(* Logix 5000 project; controller TBEN_Lx_8IOL_AOI_V0_2 vendor 1 type 14 code 176 rev 32.11; software revision 32.00; part 8 of 11 *)
(* tags used below, declared in another part *)
   Process_Input_Data : Generic_173_Words;
   Process_Output_Data : Generic_131_Words;
(* IOLService_ISDU, continued *)

ROUTINE Prescan   (* ladder *)
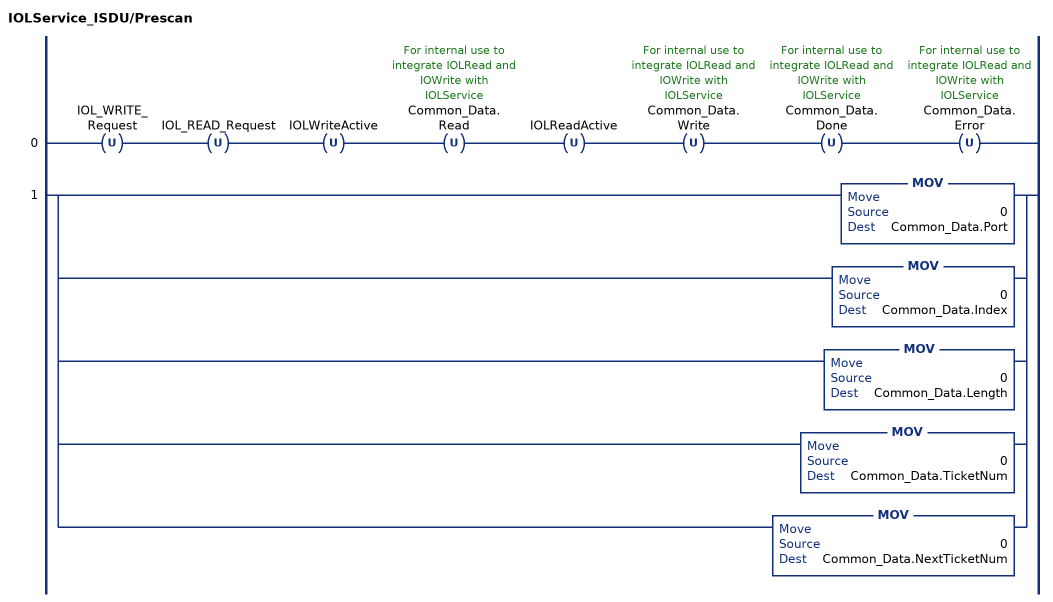
   0: OTU(IOL_WRITE_Request)OTU(IOL_READ_Request)OTU(IOLWriteActive)OTU(Common_Data.Read)OTU(IOLReadActive)OTU(Common_Data.Write)OTU(Common_Data.Done)OTU(Common_Data.Error);
   1: [MOV(0,Common_Data.Port) ,MOV(0,Common_Data.Index) ,MOV(0,Common_Data.Length) ,MOV(0,Common_Data.TicketNum) ,MOV(0,Common_Data.NextTicketNum) ];
END_ROUTINE
END_ADD_ON_INSTRUCTION

ADD_ON_INSTRUCTION TBEN_Lx_8IOL_AOI   (* revision 0.3 Unreleased, vendor Turck, ExecutePrescan *)
// AOI specific to TBEN-Lx-8IOL devices. It requires the  Input, Output, Config tags from the catalog file.
// Revision note:
// V0_1 Initial Approach
// V0_2 Cleaning Up
// V0_3 Changes to process Data
// Help:
// IOL_Service - used with Turck BL20, BL67, BLC and TBEN IOLink masters to process requests from IOL_ReadString, IOL_WriteString, IOL_ReadData and IOL_WriteData AOI's.
// Status	Description
// 0	Operation completed successfully
// 	Status = 100 - 102, Ethernet IP MSG instruction errors - check communication parameters
// 100	IOL_SendMSG completed with error, check communication parameters
// 101	IOL_RecevieMSG completed with error, check communication parameters
// 110	IOL_Service Retry Limit exceeded
// 111	Slot specified not an IOLink master
// 	Status = 1000 to 1255, no response from device, connection error
// 1016	Device not connected or Port not configured as IOLink port
// 	Status = 2000 to 2255,  device response indicates error
// 2000	Device error, no details
// 2017	Device error, Index not available
// 2018	Device error, Subindex not available
// 2032	Device error, Service temporarily not available
// 2033	Device error, Service temporarily not available - local control
// 2034	Device error, Service temporarily not available - device control
// 2035	Device error, Index not writeable
// 2048	Device error, Parameter value out of range
// 2049	Device error, Parameter value above limit
// 2050	Device error, Parameter value below limit
// 2051	Device error, Parameter value length overrun (check IOLWrite precision/string length)
// 2052	Device error, Parameter value length underrun (check IOLWrite precision/string length)
// 2053	Device error, Function not available
// 2054	Device error, Function temporarily not available
// 2064	Device error, Parameter set invalid
// 2065	Device error, Inconsistent parameter set
// 2130	Device error, Application not ready
// 	Status = 3000 to 3255,   device response indicates vendor specific error
// 3000	Vendor specific error, no details
// 3001	Vendor specific error, vendor specific error number
// 3255	Vendor specific error, vendor specific error number
// 	Status = 7000 to 7255,  IOL-M Error Codes
// 7000	Unexpected write request instead of read request
// 7001	Decode error
// 7002	Port occupied by another task
// 	Status = 8000 to 8255,  IOL-M Error Codes
// 8000	Timeout when IOL-Ds or IOL-M ports are busy
// 8001	IOL Index out of range
// 8002	Port address greater than maximum
// 8003	Port function not supported
VAR_IN_OUT
   Common_Data : Turck_IOLink_Common_Data; {required}
        .SendData[1]   // For internal use to integrate IOLRead and IOLWrite with IOLService
   IOL_Read_MSG : MESSAGE; {required}
   IOL_Write_MSG : MESSAGE; {required}
   TBEN_I_DATA : INT[173]; {required}   // Input Data from IO Block
   TBEN_O_DATA : INT[131]; {required}   // Output Data to IO Block
   TBEN_C_DATA : SINT[160]; {required}
END_VAR
VAR_OUTPUT
   DXP1_OUT : BOOL; {visible}
   DXP3_OUT : BOOL; {visible}
   DXP5_OUT : BOOL; {visible}
   DXP7_OUT : BOOL; {visible}
   IOLDevice_PORT1 : BOOL; {visible}
   IOLDevice_PORT2 : BOOL; {visible}
   IOLDevice_PORT3 : BOOL; {visible}
   IOLDevice_PORT4 : BOOL; {visible}
   IOLDevice_PORT5 : BOOL; {visible}
   IOLDevice_PORT6 : BOOL; {visible}
   IOLDevice_PORT7 : BOOL; {visible}
   IOLDevice_PORT8 : BOOL; {visible}
END_VAR
VAR_INPUT
   IOL0_DI : BOOL; {visible}
   DXP1_IN : BOOL; {visible}
   IOL2_DI : BOOL; {visible}
   DXP3_IN : BOOL; {visible}
   IOL4_DI : BOOL; {visible}
   DXP5_IN : BOOL; {visible}
   IOL6_DI : BOOL; {visible}
   DXP7_IN : BOOL; {visible}
   IOL8_DI : BOOL; {visible}
   IOL10_DI : BOOL; {visible}
   IOL12_DI : BOOL; {visible}
   IOL14_DI : BOOL; {visible}
   PORT1_Mode_IOL_or_DI : BOOL;   // 0: IO-LINK without validation 1: Port is set to DI (Power Cycle or Module Inhibit cycle require)
   PORT2_Mode_IOL_or_DI : BOOL;   // 0: IO-LINK without validation 1: Port is set to DI (Power Cycle or Module Inhibit cycle require)
   PORT3_Mode_IOL_or_DI : BOOL;   // 0: IO-LINK without validation 1: Port is set to DI (Power Cycle or Module Inhibit cycle require)
   PORT4_Mode_IOL_or_DI : BOOL;   // 0: IO-LINK without validation 1: Port is set to DI (Power Cycle or Module Inhibit cycle require)
   PORT5_Mode_IOL_or_DI : BOOL;   // 0: IO-LINK without validation 1: Port is set to DI (Power Cycle or Module Inhibit cycle require)
   PORT6_Mode_IOL_or_DI : BOOL;   // 0: IO-LINK without validation 1: Port is set to DI (Power Cycle or Module Inhibit cycle require)
   PORT7_Mode_IOL_or_DI : BOOL;   // 0: IO-LINK without validation 1: Port is set to DI (Power Cycle or Module Inhibit cycle require)
   PORT8_Mode_IOL_or_DI : BOOL;   // 0: IO-LINK without validation 1: Port is set to DI (Power Cycle or Module Inhibit cycle require)
   DisableOutput_DXP1 : BOOL;
   DisableOutput_DXP3 : BOOL;
   DisableOutput_DXP5 : BOOL;
   DisableOutput_DXP7 : BOOL;
END_VAR
VAR_OUTPUT
   Device_Restart_Required : BOOL; {visible}
END_VAR
VAR
   IOLReadActive : BOOL;
   IOLWriteActive : BOOL;
   RetryCount : DINT;
   IOL_Error_Count : DINT; {access None}
   IOLReset_ONS : BOOL; {access None}
   ER1 : BOOL; {access None}
   ER2 : BOOL; {access None}
   tempReceiveData : SINT[255]; {access None}
   Generate_Status : BOOL; {access None}
   ABS_RD_0 : INT; {access None}
   ABS_RD_1 : INT; {access None}
   ABS_RD_2 : INT; {access None}
   ABS_RD_3 : INT; {access None}
   tempSendData : SINT[145]; {access None}
   IOL_READ_Request : BOOL; {access None}
   IOL_WRITE_Request : BOOL; {access None}
   StartupDone : BOOL; {access None}
   Done : BOOL; {access None}
   Error : BOOL; {access None}
   Active : BOOL; {access None}
   Pending : BOOL; {access None}
   Pending_or_Active : BOOL; {access None}
   StartupCount : SINT; {access None}
   DoneCount : SINT; {access None}
   MyTicketNum : INT; {access None}
   Update_Data : BOOL; {access None}
   Read_ONS : BOOL; {access None}
   ReadRequest : BOOL; {access None}
   Prev_Input_Data_Valids : INT; {access None}
   Status : DINT; {access None}
   ErrorCount : DINT; {access None}
   PIDV_Delay : TIMER := (PRE := 1000); {access None}
   TimeDelay : TIMER := (PRE := 500); {access None}
END_VAR

ROUTINE Logic   (* ladder *)
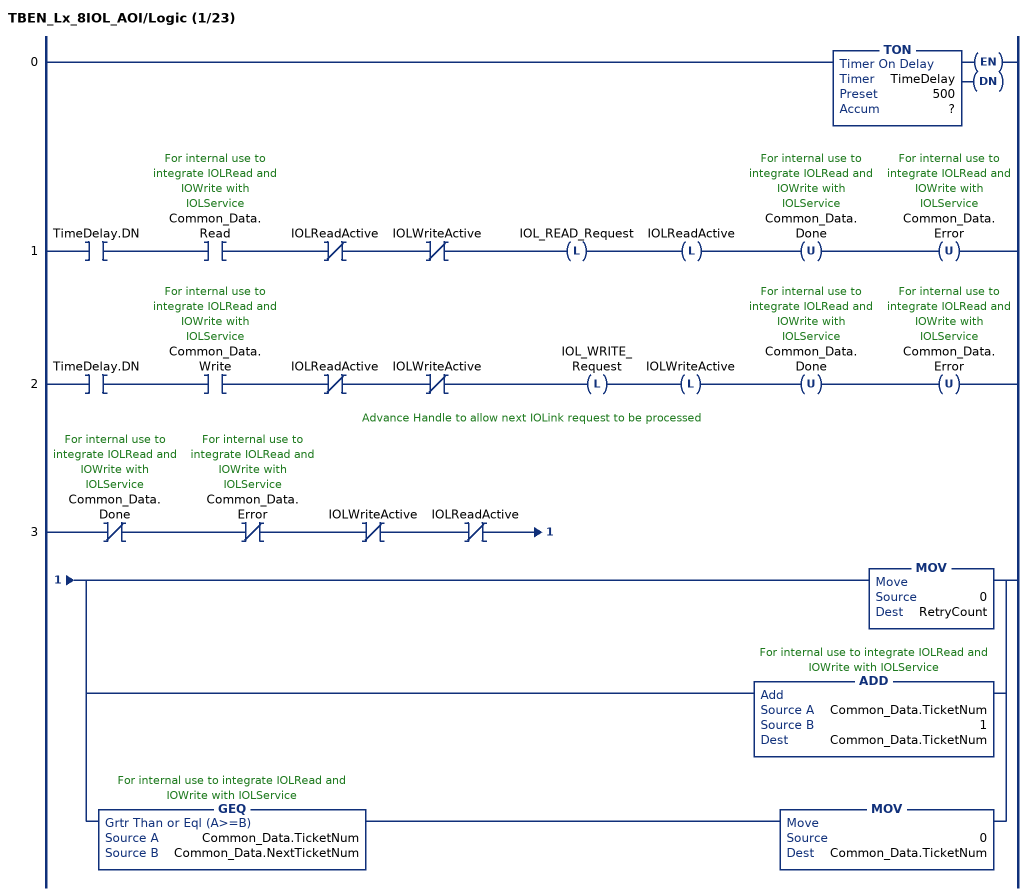
   0: TON(TimeDelay,?,?);
   1: XIC(TimeDelay.DN)XIC(Common_Data.Read)XIO(IOLReadActive)XIO(IOLWriteActive)OTL(IOL_READ_Request)OTL(IOLReadActive)OTU(Common_Data.Done)OTU(Common_Data.Error);
   2: XIC(TimeDelay.DN)XIC(Common_Data.Write)XIO(IOLReadActive)XIO(IOLWriteActive)OTL(IOL_WRITE_Request)OTL(IOLWriteActive)OTU(Common_Data.Done)OTU(Common_Data.Error);
   // Advance Handle to allow next IOLink request to be processed
   3: XIO(Common_Data.Done)XIO(Common_Data.Error)XIO(IOLWriteActive)XIO(IOLReadActive)[MOV(0,RetryCount) ,ADD(Common_Data.TicketNum,1,Common_Data.TicketNum) ,GEQ(Common_Data.TicketNum,Common_Data.NextTicketNum) MOV(0,Common_Data.TicketNum) ];
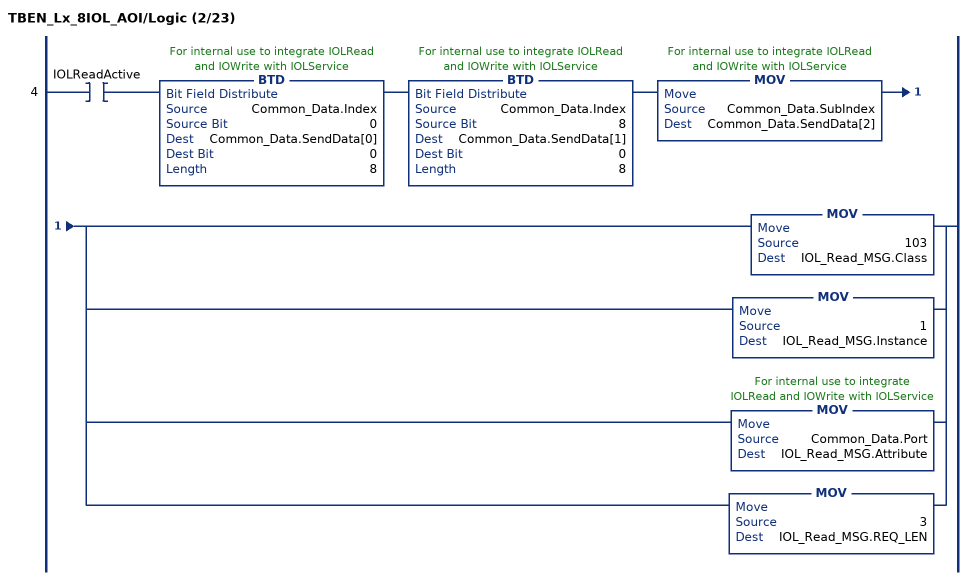
   4: XIC(IOLReadActive)BTD(Common_Data.Index,0,Common_Data.SendData[0],0,8)BTD(Common_Data.Index,8,Common_Data.SendData[1],0,8)MOV(Common_Data.SubIndex,Common_Data.SendData[2])[MOV(103,IOL_Read_MSG.Class) ,MOV(1,IOL_Read_MSG.Instance) ,MOV(Common_Data.Port,IOL_Read_MSG.Attribute) ,MOV(3,IOL_Read_MSG.REQ_LEN) ];
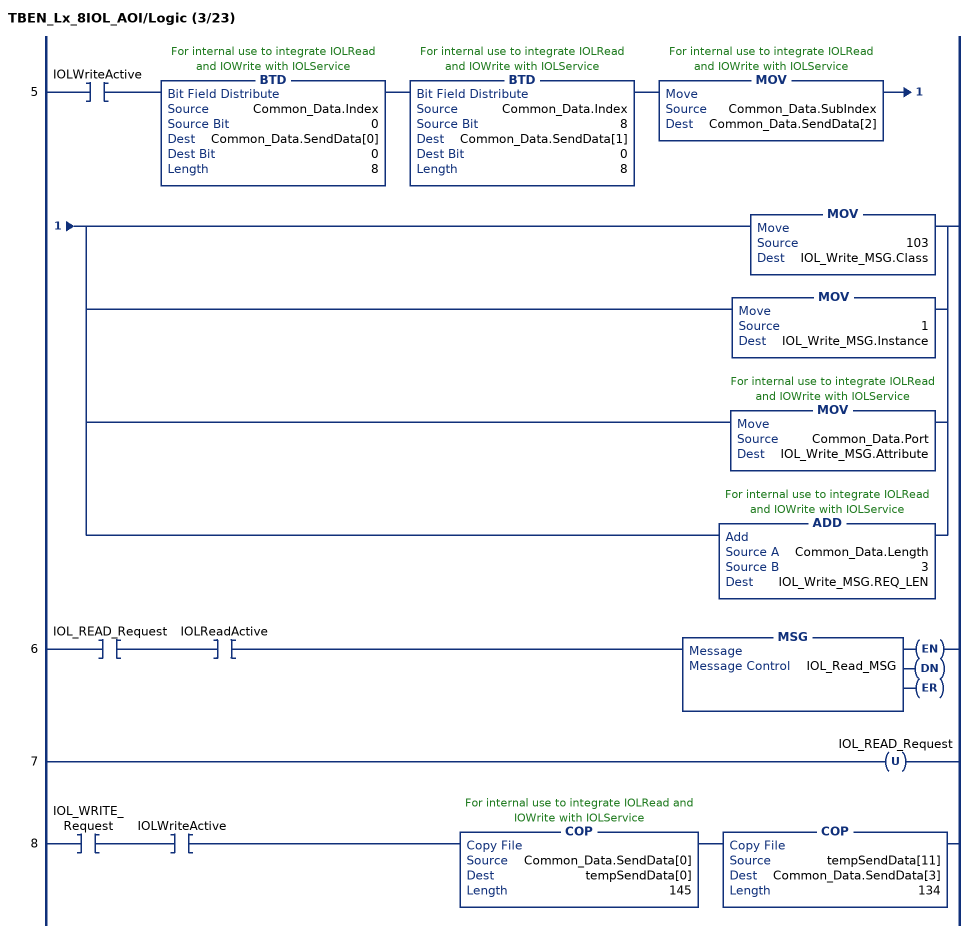
   5: XIC(IOLWriteActive)BTD(Common_Data.Index,0,Common_Data.SendData[0],0,8)BTD(Common_Data.Index,8,Common_Data.SendData[1],0,8)MOV(Common_Data.SubIndex,Common_Data.SendData[2])[MOV(103,IOL_Write_MSG.Class) ,MOV(1,IOL_Write_MSG.Instance) ,MOV(Common_Data.Port,IOL_Write_MSG.Attribute) ,ADD(Common_Data.Length,3,IOL_Write_MSG.REQ_LEN) ];
   6: XIC(IOL_READ_Request)XIC(IOLReadActive)MSG(IOL_Read_MSG);
   7: OTU(IOL_READ_Request);
   8: XIC(IOL_WRITE_Request)XIC(IOLWriteActive)COP(Common_Data.SendData[0],tempSendData[0],145)COP(tempSendData[11],Common_Data.SendData[3],134);
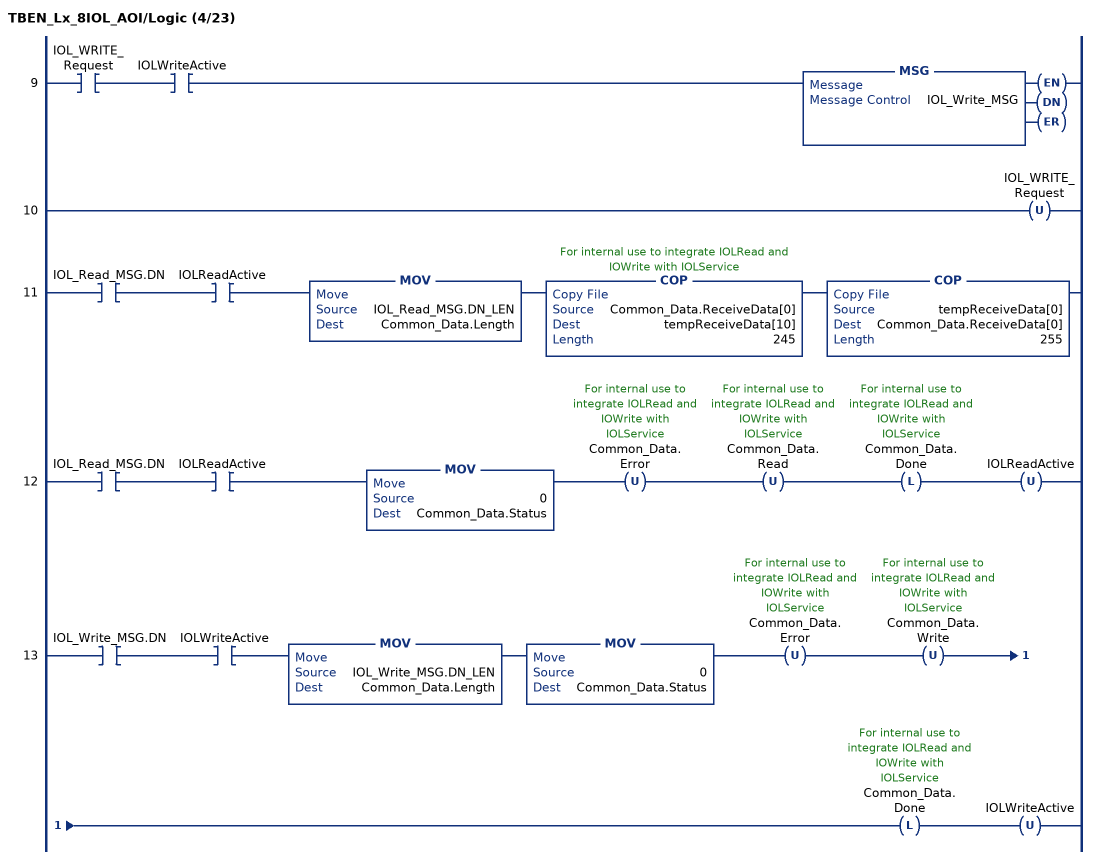
   9: XIC(IOL_WRITE_Request)XIC(IOLWriteActive)MSG(IOL_Write_MSG);
   10: OTU(IOL_WRITE_Request);
   11: XIC(IOL_Read_MSG.DN)XIC(IOLReadActive)MOV(IOL_Read_MSG.DN_LEN,Common_Data.Length)COP(Common_Data.ReceiveData[0],tempReceiveData[10],245)COP(tempReceiveData[0],Common_Data.ReceiveData[0],255);
   12: XIC(IOL_Read_MSG.DN)XIC(IOLReadActive)MOV(0,Common_Data.Status)OTU(Common_Data.Error)OTU(Common_Data.Read)OTL(Common_Data.Done)OTU(IOLReadActive);
   13: XIC(IOL_Write_MSG.DN)XIC(IOLWriteActive)MOV(IOL_Write_MSG.DN_LEN,Common_Data.Length)MOV(0,Common_Data.Status)OTU(Common_Data.Error)OTU(Common_Data.Write)OTL(Common_Data.Done)OTU(IOLWriteActive);
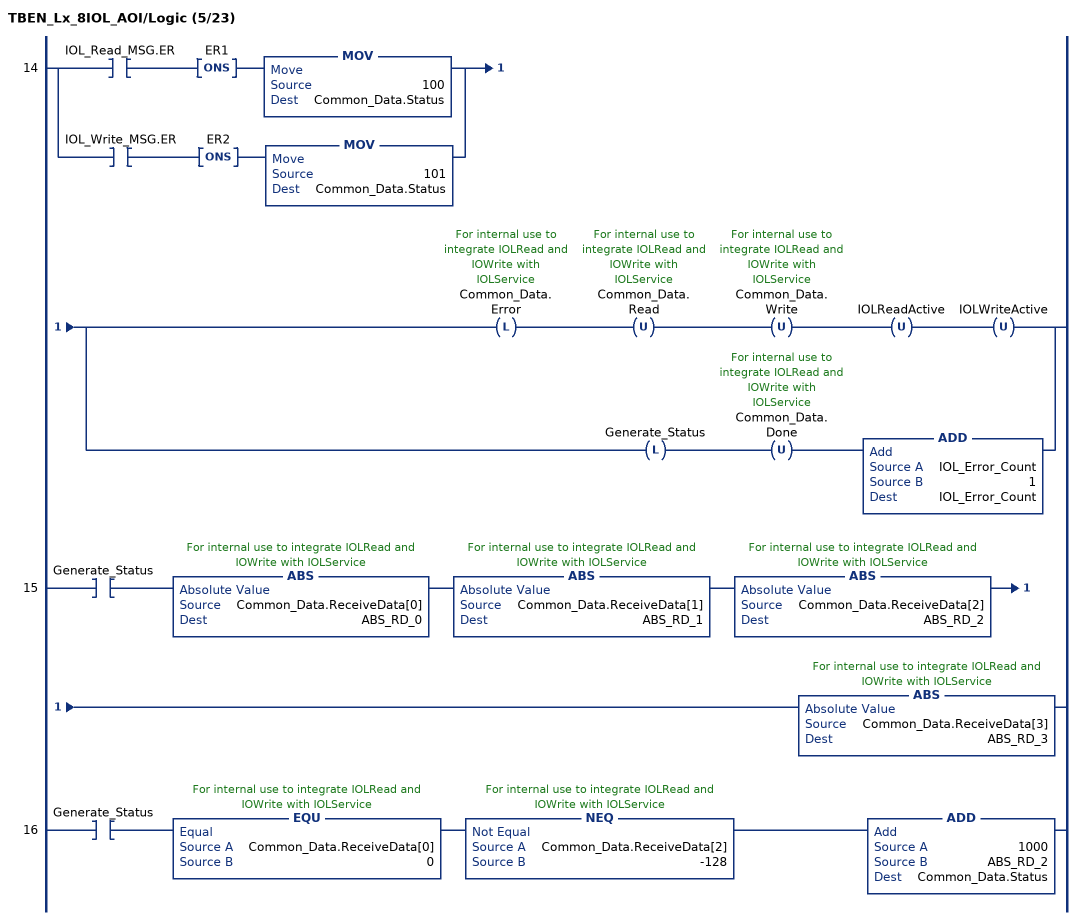
   14: [XIC(IOL_Read_MSG.ER) ONS(ER1) MOV(100,Common_Data.Status) ,XIC(IOL_Write_MSG.ER) ONS(ER2) MOV(101,Common_Data.Status) ][OTL(Common_Data.Error) OTU(Common_Data.Read) OTU(Common_Data.Write) OTU(IOLReadActive) OTU(IOLWriteActive) ,OTL(Generate_Status) OTU(Common_Data.Done) ADD(IOL_Error_Count,1,IOL_Error_Count) ];
   15: XIC(Generate_Status)ABS(Common_Data.ReceiveData[0],ABS_RD_0)ABS(Common_Data.ReceiveData[1],ABS_RD_1)ABS(Common_Data.ReceiveData[2],ABS_RD_2)ABS(Common_Data.ReceiveData[3],ABS_RD_3);
   16: XIC(Generate_Status)EQU(Common_Data.ReceiveData[0],0)NEQ(Common_Data.ReceiveData[2],-128)ADD(1000,ABS_RD_2,Common_Data.Status);
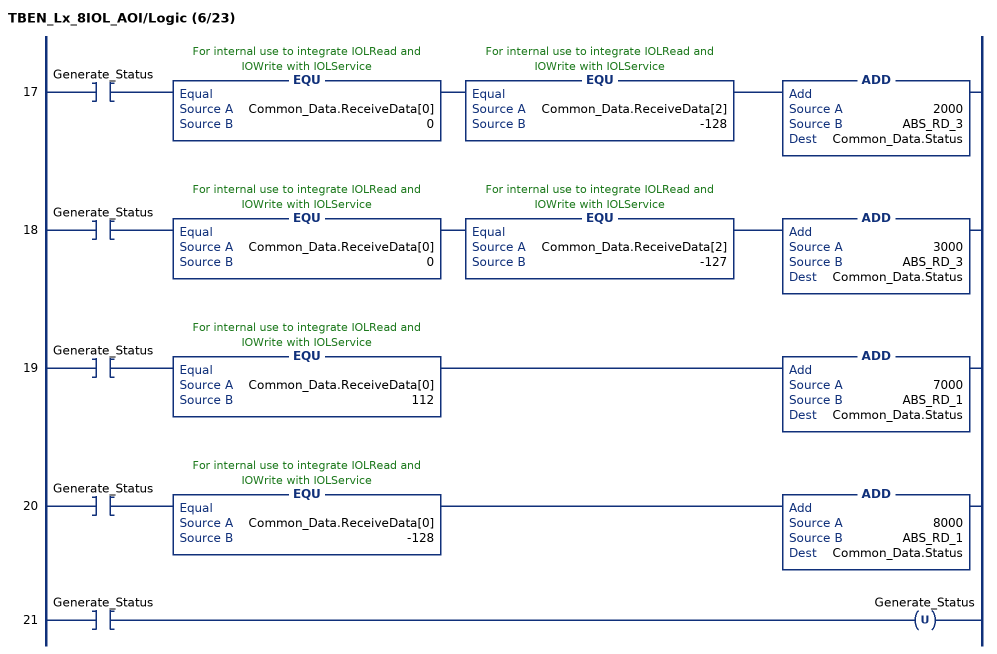
   17: XIC(Generate_Status)EQU(Common_Data.ReceiveData[0],0)EQU(Common_Data.ReceiveData[2],-128)ADD(2000,ABS_RD_3,Common_Data.Status);
   18: XIC(Generate_Status)EQU(Common_Data.ReceiveData[0],0)EQU(Common_Data.ReceiveData[2],-127)ADD(3000,ABS_RD_3,Common_Data.Status);
   19: XIC(Generate_Status)EQU(Common_Data.ReceiveData[0],112)ADD(7000,ABS_RD_1,Common_Data.Status);
   20: XIC(Generate_Status)EQU(Common_Data.ReceiveData[0],-128)ADD(8000,ABS_RD_1,Common_Data.Status);
   21: XIC(Generate_Status)OTU(Generate_Status);
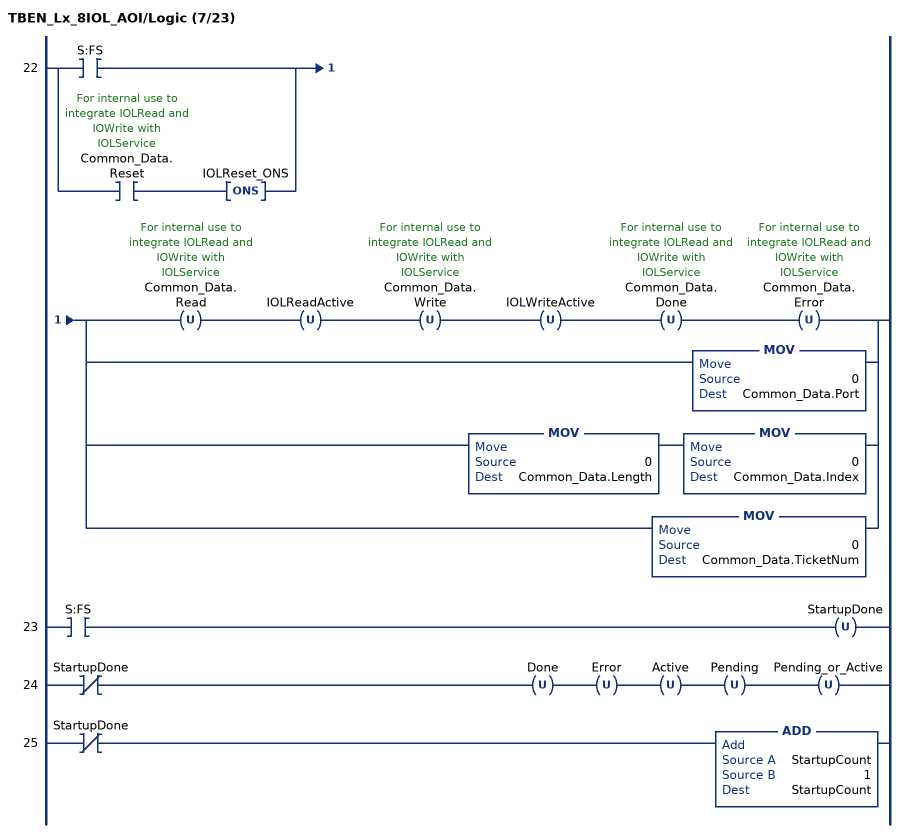
   22: [XIC(S:FS) ,XIC(Common_Data.Reset) ONS(IOLReset_ONS) ][OTU(Common_Data.Read) OTU(IOLReadActive) OTU(Common_Data.Write) OTU(IOLWriteActive) OTU(Common_Data.Done) OTU(Common_Data.Error) ,MOV(0,Common_Data.Port) ,MOV(0,Common_Data.Length) MOV(0,Common_Data.Index) ,MOV(0,Common_Data.TicketNum) ];
   23: XIC(S:FS)OTU(StartupDone);
   24: XIO(StartupDone)OTU(Done)OTU(Error)OTU(Active)OTU(Pending)OTU(Pending_or_Active);
   25: XIO(StartupDone)ADD(StartupCount,1,StartupCount);
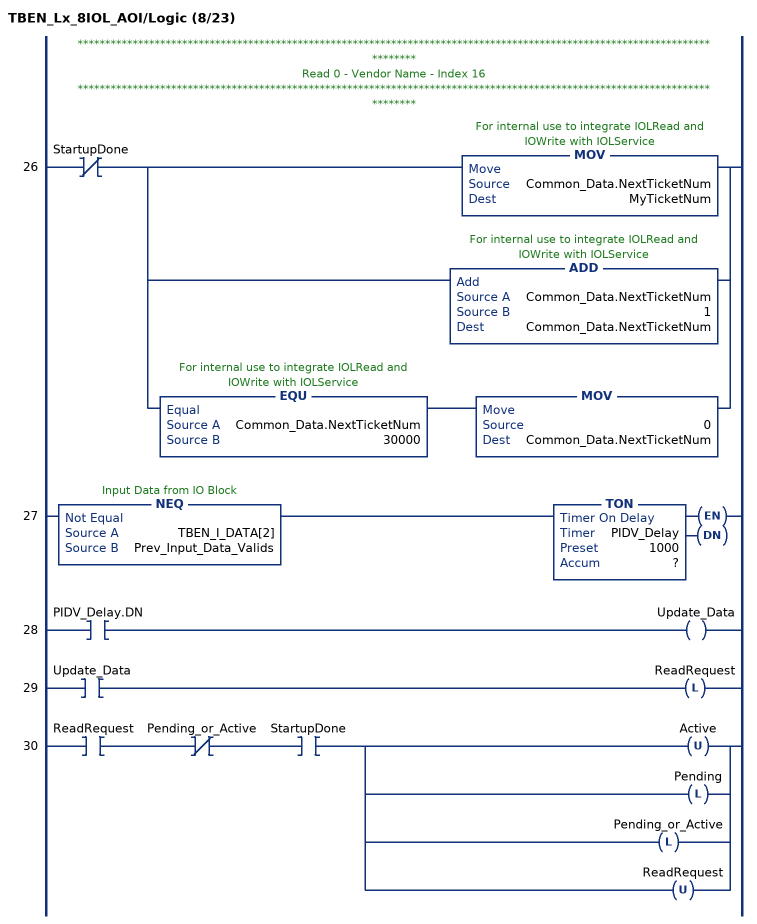
   // ***************************************************************************************************************************
   // Read 0 - Vendor Name - Index 16
   // ***************************************************************************************************************************
   26: XIO(StartupDone)[MOV(Common_Data.NextTicketNum,MyTicketNum) ,ADD(Common_Data.NextTicketNum,1,Common_Data.NextTicketNum) ,EQU(Common_Data.NextTicketNum,30000) MOV(0,Common_Data.NextTicketNum) ];
   27: NEQ(TBEN_I_DATA[2],Prev_Input_Data_Valids)TON(PIDV_Delay,?,?);
   28: XIC(PIDV_Delay.DN)OTE(Update_Data);
   29: XIC(Update_Data)OTL(ReadRequest);
   30: XIC(ReadRequest)XIO(Pending_or_Active)XIC(StartupDone)[OTU(Active) ,OTL(Pending) ,OTL(Pending_or_Active) ,OTU(ReadRequest) ];
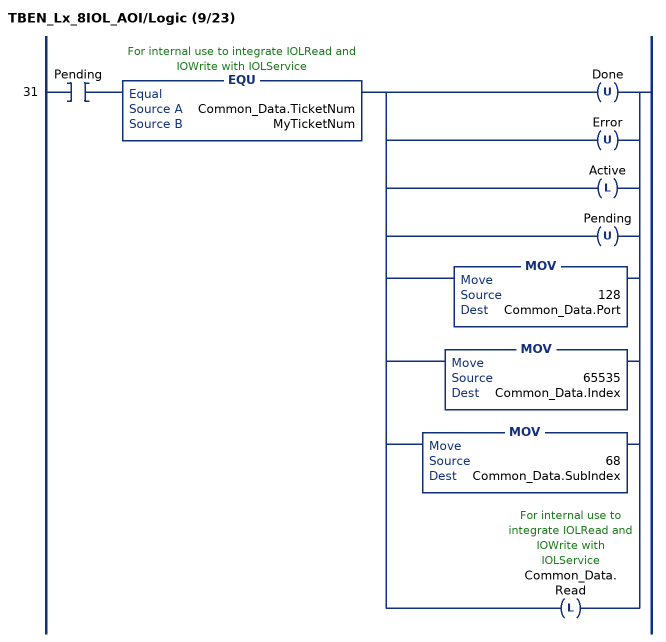
   31: XIC(Pending)EQU(Common_Data.TicketNum,MyTicketNum)[OTU(Done) ,OTU(Error) ,OTL(Active) ,OTU(Pending) ,MOV(128,Common_Data.Port) ,MOV(65535,Common_Data.Index) ,MOV(68,Common_Data.SubIndex) ,OTL(Common_Data.Read) ];
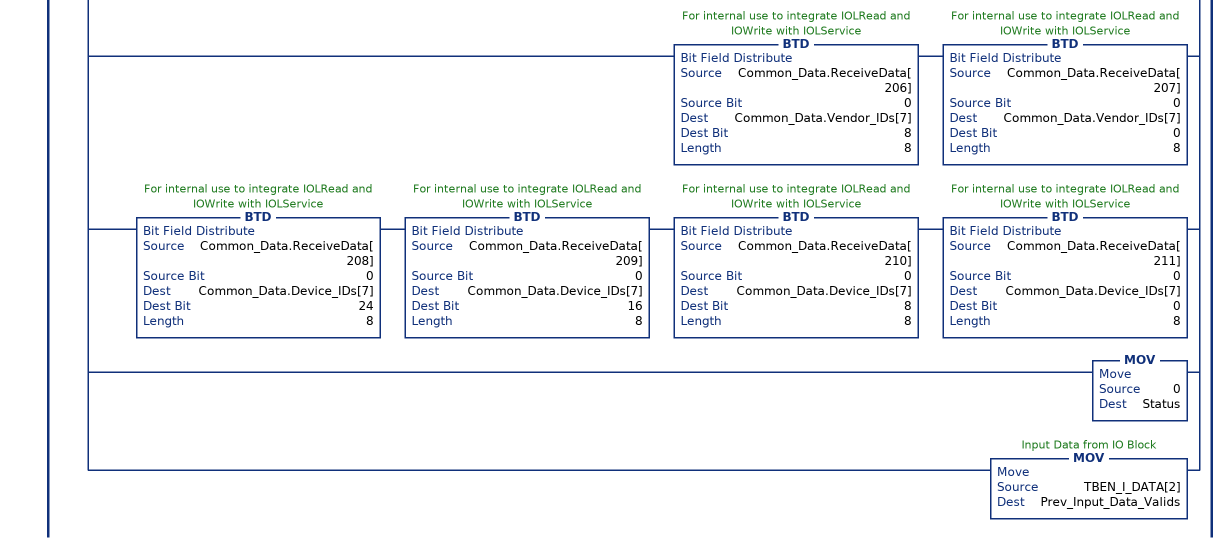
   // Get VIDs/DIDs for evry port.
   32: XIC(Active)XIC(Common_Data.Done)[OTL(Done) ,ADD(DoneCount,1,DoneCount) ,OTU(Error) ,OTU(Active) ,OTU(Pending) ,OTU(Pending_or_Active) ,OTU(Common_Data.Done) ,BTD(Common_Data.ReceiveData[10],0,Common_Data.Vendor_IDs[0],8,8) BTD(Common_Data.ReceiveData[11],0,Common_Data.Vendor_IDs[0],0,8) ,BTD(Common_Data.ReceiveData[12],0,Common_Data.Device_IDs[0],24,8) BTD(Common_Data.ReceiveData[13],0,Common_Data.Device_IDs[0],16,8) BTD(Common_Data.ReceiveData[14],0,Common_Data.Device_IDs[0],8,8) BTD(Common_Data.ReceiveData[15],0,Common_Data.Device_IDs[0],0,8) ,BTD(Common_Data.ReceiveData[38],0,Common_Data.Vendor_IDs[1],8,8) BTD(Common_Data.ReceiveData[39],0,Common_Data.Vendor_IDs[1],0,8) ,BTD(Common_Data.ReceiveData[40],0,Common_Data.Device_IDs[1],24,8) BTD(Common_Data.ReceiveData[41],0,Common_Data.Device_IDs[1],16,8) BTD(Common_Data.ReceiveData[42],0,Common_Data.Device_IDs[1],8,8) BTD(Common_Data.ReceiveData[43],0,Common_Data.Device_IDs[1],0,8) ,BTD(Common_Data.ReceiveData[66],0,Common_Data.Vendor_IDs[2],8,8) BTD(Common_Data.ReceiveData[67],0,Common_Data.Vendor_IDs[2],0,8) ,BTD(Common_Data.ReceiveData[68],0,Common_Data.Device_IDs[2],24,8) BTD(Common_Data.ReceiveData[69],0,Common_Data.Device_IDs[2],16,8) BTD(Common_Data.ReceiveData[70],0,Common_Data.Device_IDs[2],8,8) BTD(Common_Data.ReceiveData[71],0,Common_Data.Device_IDs[2],0,8) ,BTD(Common_Data.ReceiveData[94],0,Common_Data.Vendor_IDs[3],8,8) BTD(Common_Data.ReceiveData[95],0,Common_Data.Vendor_IDs[3],0,8) ,BTD(Common_Data.ReceiveData[96],0,Common_Data.Device_IDs[3],24,8) BTD(Common_Data.ReceiveData[97],0,Common_Data.Device_IDs[3],16,8) BTD(Common_Data.ReceiveData[98],0,Common_Data.Device_IDs[3],8,8) BTD(Common_Data.ReceiveData[99],0,Common_Data.Device_IDs[3],0,8) ,BTD(Common_Data.ReceiveData[122],0,Common_Data.Vendor_IDs[4],8,8) BTD(Common_Data.ReceiveData[123],0,Common_Data.Vendor_IDs[4],0,8) ,BTD(Common_Data.ReceiveData[124],0,Common_Data.Device_IDs[4],24,8) BTD(Common_Data.ReceiveData[125],0,Common_Data.Device_IDs[4],16,8) BTD(Common_Data.ReceiveData[126],0,Common_Data.Device_IDs[4],8,8) BTD(Common_Data.ReceiveData[127],0,Common_Data.Device_IDs[4],0,8) ,BTD(Common_Data.ReceiveData[150],0,Common_Data.Vendor_IDs[5],8,8) BTD(Common_Data.ReceiveData[151],0,Common_Data.Vendor_IDs[5],0,8) ,BTD(Common_Data.ReceiveData[152],0,Common_Data.Device_IDs[5],24,8) BTD(Common_Data.ReceiveData[153],0,Common_Data.Device_IDs[5],16,8) BTD(Common_Data.ReceiveData[154],0,Common_Data.Device_IDs[5],8,8) BTD(Common_Data.ReceiveData[155],0,Common_Data.Device_IDs[5],0,8) ,BTD(Common_Data.ReceiveData[178],0,Common_Data.Vendor_IDs[6],8,8) BTD(Common_Data.ReceiveData[179],0,Common_Data.Vendor_IDs[6],0,8) ,BTD(Common_Data.ReceiveData[180],0,Common_Data.Device_IDs[6],24,8) BTD(Common_Data.ReceiveData[181],0,Common_Data.Device_IDs[6],16,8) BTD(Common_Data.ReceiveData[182],0,Common_Data.Device_IDs[6],8,8) BTD(Common_Data.ReceiveData[183],0,Common_Data.Device_IDs[6],0,8) ,BTD(Common_Data.ReceiveData[206],0,Common_Data.Vendor_IDs[7],8,8) BTD(Common_Data.ReceiveData[207],0,Common_Data.Vendor_IDs[7],0,8) ,BTD(Common_Data.ReceiveData[208],0,Common_Data.Device_IDs[7],24,8) BTD(Common_Data.ReceiveData[209],0,Common_Data.Device_IDs[7],16,8) BTD(Common_Data.ReceiveData[210],0,Common_Data.Device_IDs[7],8,8) BTD(Common_Data.ReceiveData[211],0,Common_Data.Device_IDs[7],0,8) ,MOV(0,Status) ,MOV(TBEN_I_DATA[2],Prev_Input_Data_Valids) ];
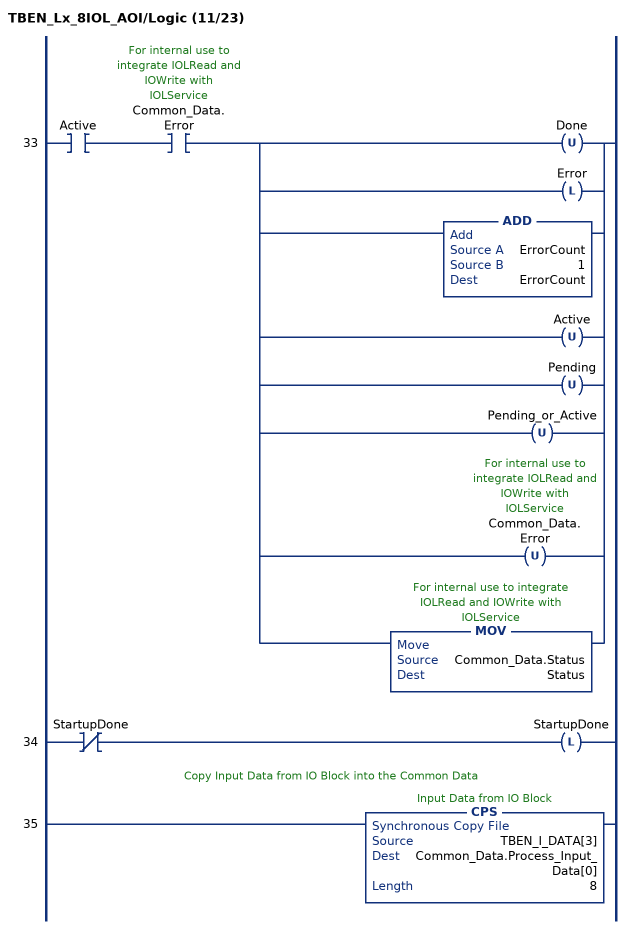
   33: XIC(Active)XIC(Common_Data.Error)[OTU(Done) ,OTL(Error) ,ADD(ErrorCount,1,ErrorCount) ,OTU(Active) ,OTU(Pending) ,OTU(Pending_or_Active) ,OTU(Common_Data.Error) ,MOV(Common_Data.Status,Status) ];
   34: XIO(StartupDone)OTL(StartupDone);
   // Copy Input Data from IO Block into the Common Data
   35: CPS(TBEN_I_DATA[3],Common_Data.Process_Input_Data[0],8);
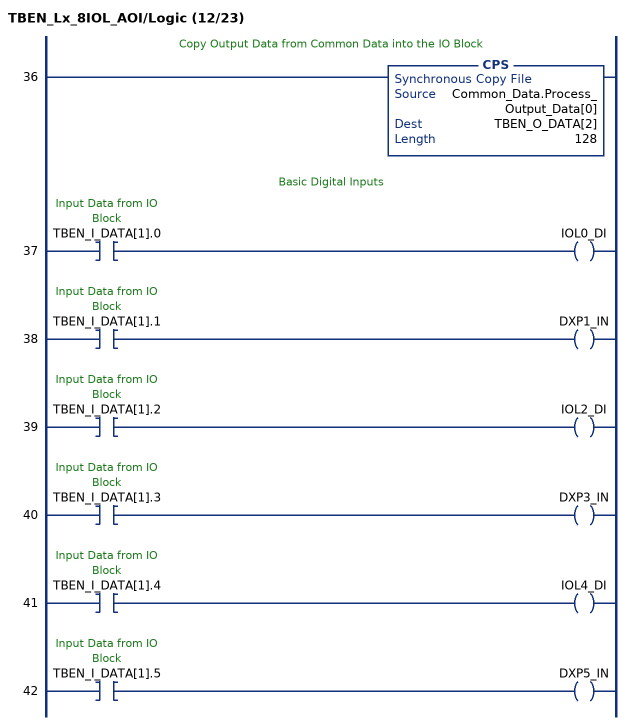
   // Copy Output Data from Common Data into the IO Block
   36: CPS(Common_Data.Process_Output_Data[0],TBEN_O_DATA[2],128);
   // Basic Digital Inputs
   37: XIC(TBEN_I_DATA[1].0)OTE(IOL0_DI);
   38: XIC(TBEN_I_DATA[1].1)OTE(DXP1_IN);
   39: XIC(TBEN_I_DATA[1].2)OTE(IOL2_DI);
   40: XIC(TBEN_I_DATA[1].3)OTE(DXP3_IN);
   41: XIC(TBEN_I_DATA[1].4)OTE(IOL4_DI);
   42: XIC(TBEN_I_DATA[1].5)OTE(DXP5_IN);
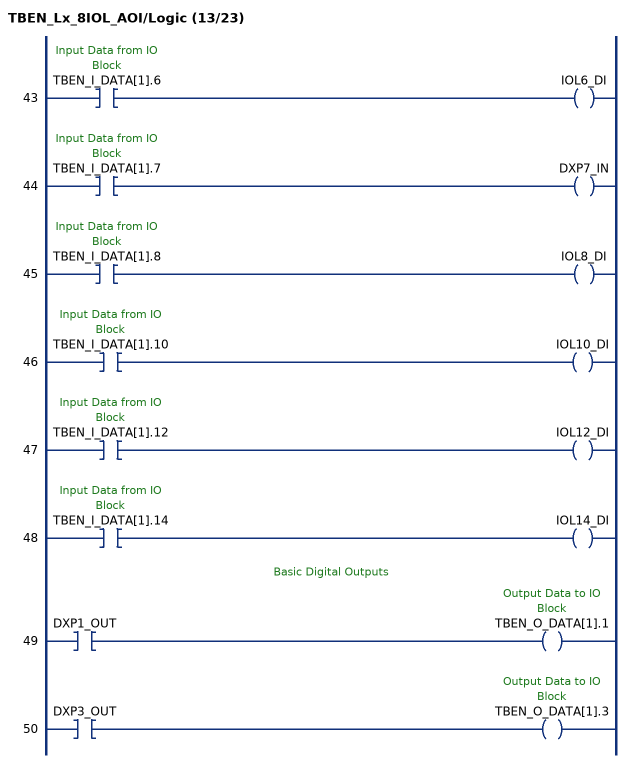
   43: XIC(TBEN_I_DATA[1].6)OTE(IOL6_DI);
   44: XIC(TBEN_I_DATA[1].7)OTE(DXP7_IN);
   45: XIC(TBEN_I_DATA[1].8)OTE(IOL8_DI);
   46: XIC(TBEN_I_DATA[1].10)OTE(IOL10_DI);
   47: XIC(TBEN_I_DATA[1].12)OTE(IOL12_DI);
   48: XIC(TBEN_I_DATA[1].14)OTE(IOL14_DI);
   // Basic Digital Outputs
   49: XIC(DXP1_OUT)OTE(TBEN_O_DATA[1].1);
   50: XIC(DXP3_OUT)OTE(TBEN_O_DATA[1].3);
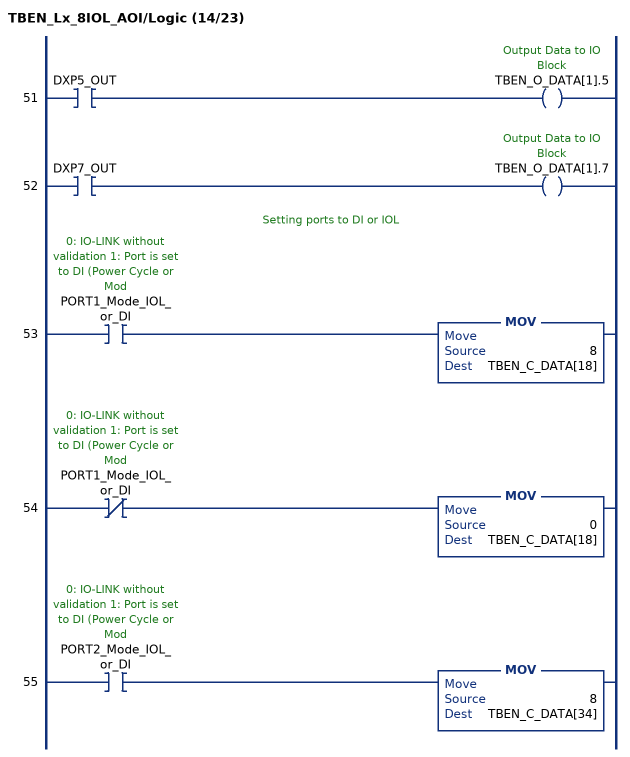
   51: XIC(DXP5_OUT)OTE(TBEN_O_DATA[1].5);
   52: XIC(DXP7_OUT)OTE(TBEN_O_DATA[1].7);
   // Setting ports to DI or IOL
   53: XIC(PORT1_Mode_IOL_or_DI)MOV(8,TBEN_C_DATA[18]);
   54: XIO(PORT1_Mode_IOL_or_DI)MOV(0,TBEN_C_DATA[18]);
   55: XIC(PORT2_Mode_IOL_or_DI)MOV(8,TBEN_C_DATA[34]);
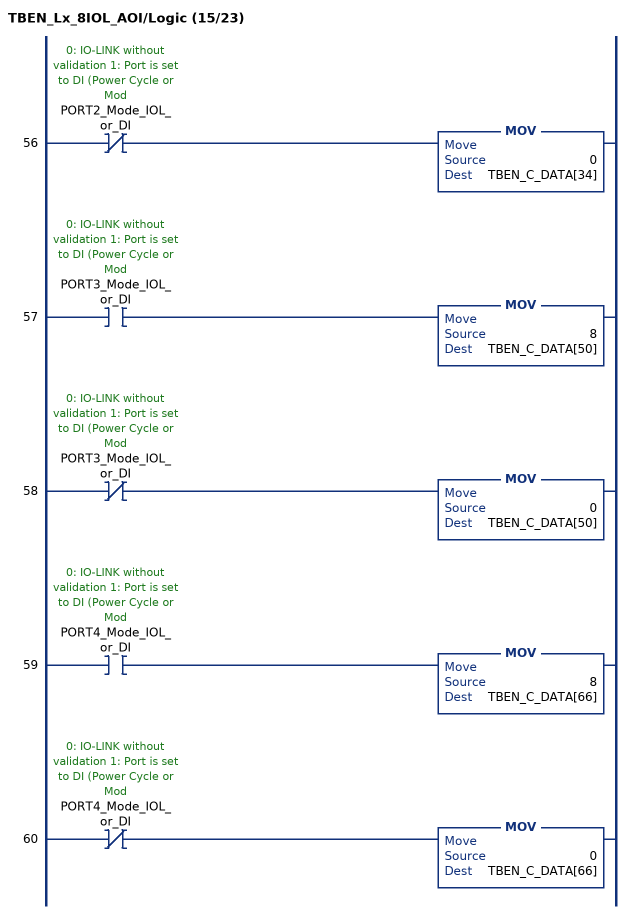
   56: XIO(PORT2_Mode_IOL_or_DI)MOV(0,TBEN_C_DATA[34]);
   57: XIC(PORT3_Mode_IOL_or_DI)MOV(8,TBEN_C_DATA[50]);
   58: XIO(PORT3_Mode_IOL_or_DI)MOV(0,TBEN_C_DATA[50]);
   59: XIC(PORT4_Mode_IOL_or_DI)MOV(8,TBEN_C_DATA[66]);
   60: XIO(PORT4_Mode_IOL_or_DI)MOV(0,TBEN_C_DATA[66]);
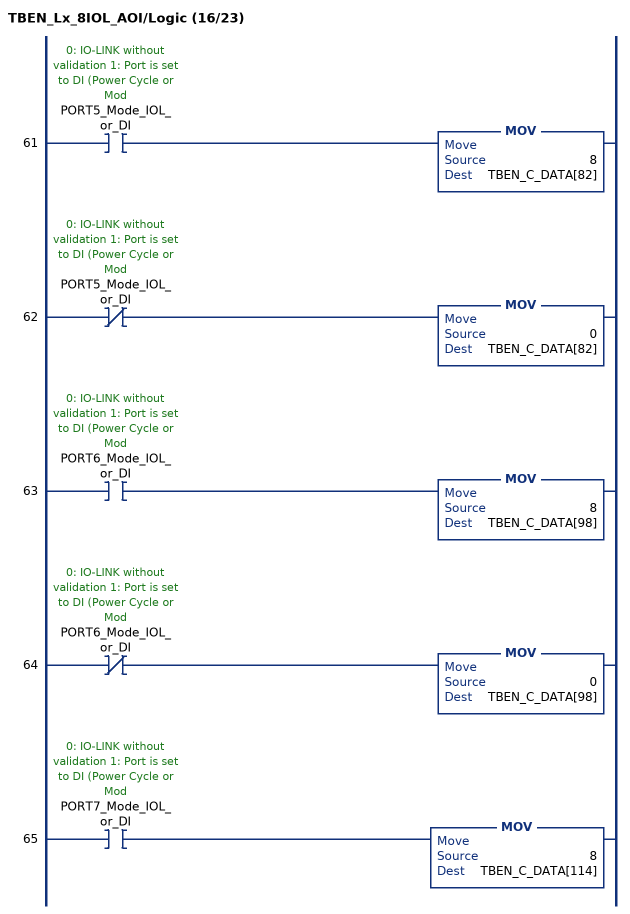
   61: XIC(PORT5_Mode_IOL_or_DI)MOV(8,TBEN_C_DATA[82]);
   62: XIO(PORT5_Mode_IOL_or_DI)MOV(0,TBEN_C_DATA[82]);
   63: XIC(PORT6_Mode_IOL_or_DI)MOV(8,TBEN_C_DATA[98]);
   64: XIO(PORT6_Mode_IOL_or_DI)MOV(0,TBEN_C_DATA[98]);
   65: XIC(PORT7_Mode_IOL_or_DI)MOV(8,TBEN_C_DATA[114]);
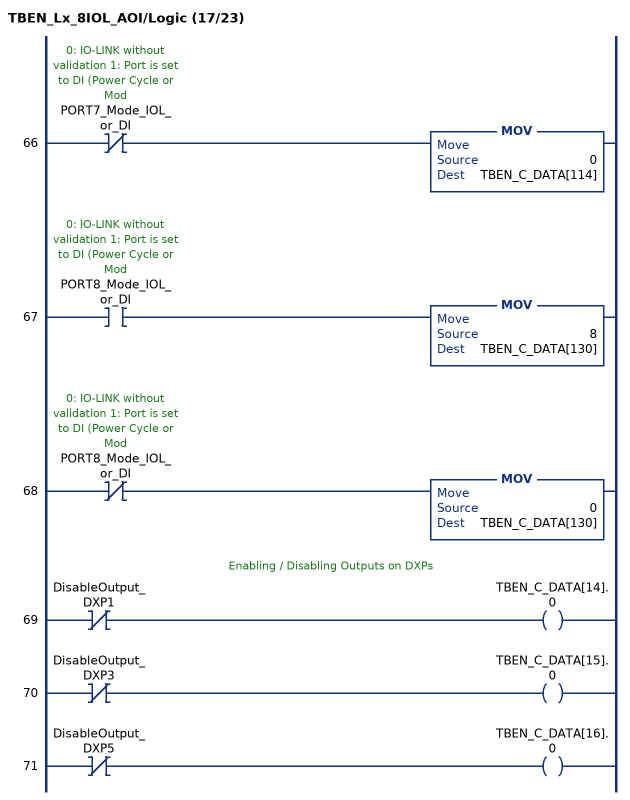
   66: XIO(PORT7_Mode_IOL_or_DI)MOV(0,TBEN_C_DATA[114]);
   67: XIC(PORT8_Mode_IOL_or_DI)MOV(8,TBEN_C_DATA[130]);
   68: XIO(PORT8_Mode_IOL_or_DI)MOV(0,TBEN_C_DATA[130]);
   // Enabling / Disabling Outputs on DXPs
   69: XIO(DisableOutput_DXP1)OTE(TBEN_C_DATA[14].0);
   70: XIO(DisableOutput_DXP3)OTE(TBEN_C_DATA[15].0);
   71: XIO(DisableOutput_DXP5)OTE(TBEN_C_DATA[16].0);
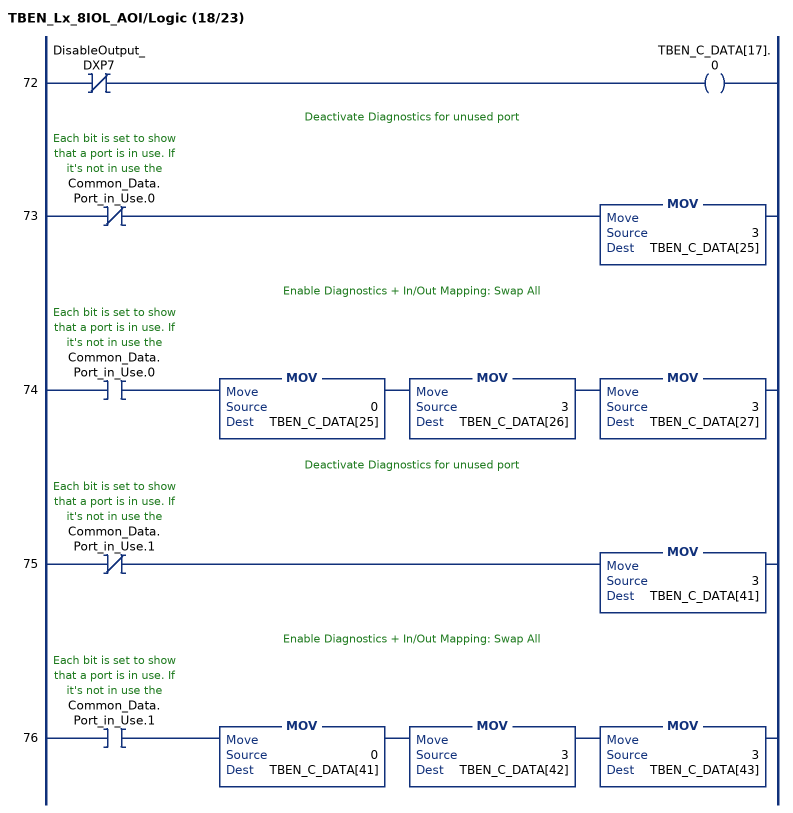
   72: XIO(DisableOutput_DXP7)OTE(TBEN_C_DATA[17].0);
   // Deactivate Diagnostics for unused port
   73: XIO(Common_Data.Port_in_Use.0)MOV(3,TBEN_C_DATA[25]);
   // Enable Diagnostics + In/Out Mapping: Swap All
   74: XIC(Common_Data.Port_in_Use.0)MOV(0,TBEN_C_DATA[25])MOV(3,TBEN_C_DATA[26])MOV(3,TBEN_C_DATA[27]);
   // Deactivate Diagnostics for unused port
   75: XIO(Common_Data.Port_in_Use.1)MOV(3,TBEN_C_DATA[41]);
   // Enable Diagnostics + In/Out Mapping: Swap All
   76: XIC(Common_Data.Port_in_Use.1)MOV(0,TBEN_C_DATA[41])MOV(3,TBEN_C_DATA[42])MOV(3,TBEN_C_DATA[43]);
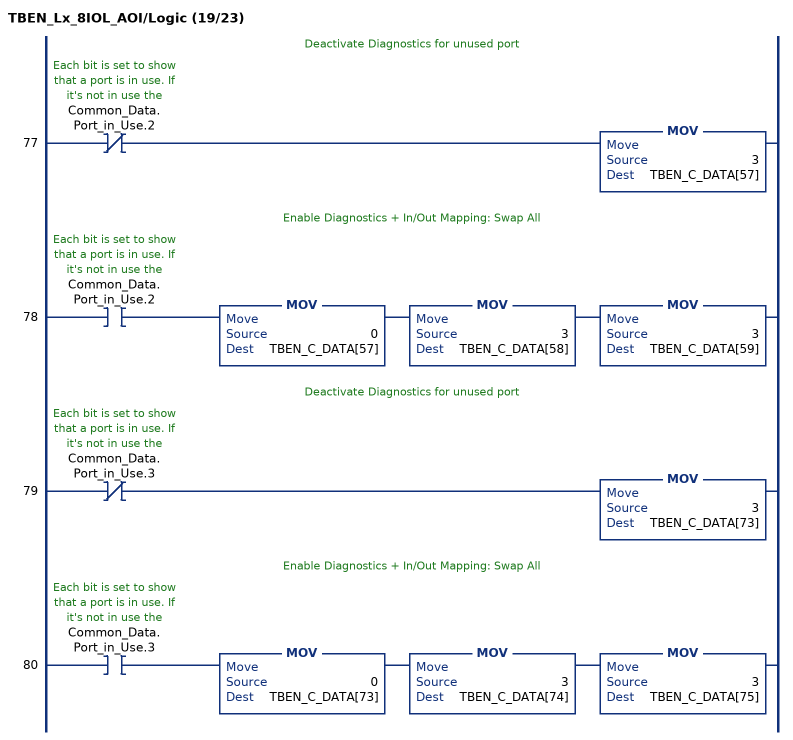
   // Deactivate Diagnostics for unused port
   77: XIO(Common_Data.Port_in_Use.2)MOV(3,TBEN_C_DATA[57]);
   // Enable Diagnostics + In/Out Mapping: Swap All
   78: XIC(Common_Data.Port_in_Use.2)MOV(0,TBEN_C_DATA[57])MOV(3,TBEN_C_DATA[58])MOV(3,TBEN_C_DATA[59]);
   // Deactivate Diagnostics for unused port
   79: XIO(Common_Data.Port_in_Use.3)MOV(3,TBEN_C_DATA[73]);
   // Enable Diagnostics + In/Out Mapping: Swap All
   80: XIC(Common_Data.Port_in_Use.3)MOV(0,TBEN_C_DATA[73])MOV(3,TBEN_C_DATA[74])MOV(3,TBEN_C_DATA[75]);
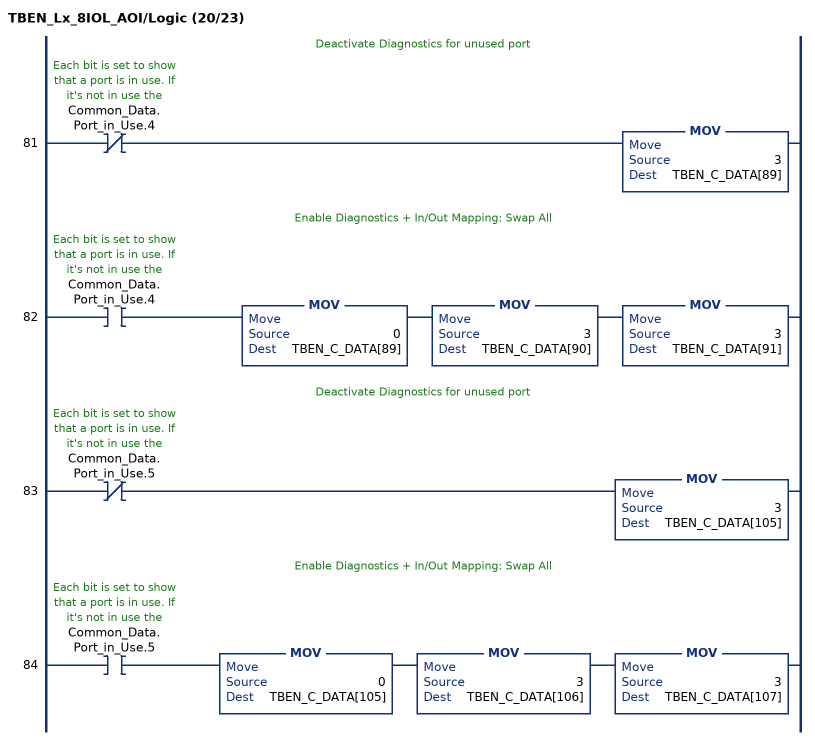
   // Deactivate Diagnostics for unused port
   81: XIO(Common_Data.Port_in_Use.4)MOV(3,TBEN_C_DATA[89]);
   // Enable Diagnostics + In/Out Mapping: Swap All
   82: XIC(Common_Data.Port_in_Use.4)MOV(0,TBEN_C_DATA[89])MOV(3,TBEN_C_DATA[90])MOV(3,TBEN_C_DATA[91]);
   // Deactivate Diagnostics for unused port
   83: XIO(Common_Data.Port_in_Use.5)MOV(3,TBEN_C_DATA[105]);
   // Enable Diagnostics + In/Out Mapping: Swap All
   84: XIC(Common_Data.Port_in_Use.5)MOV(0,TBEN_C_DATA[105])MOV(3,TBEN_C_DATA[106])MOV(3,TBEN_C_DATA[107]);
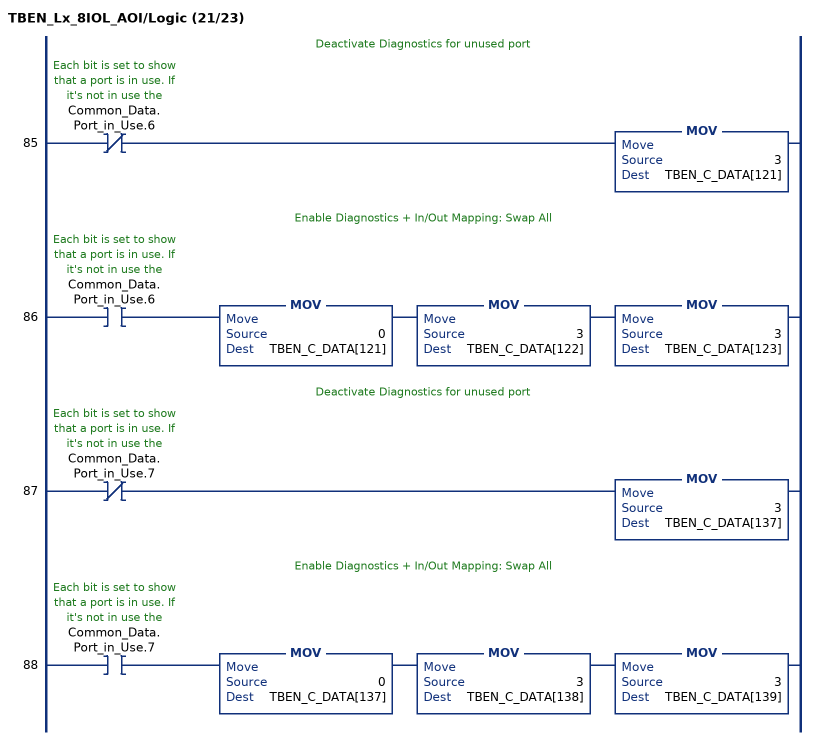
   // Deactivate Diagnostics for unused port
   85: XIO(Common_Data.Port_in_Use.6)MOV(3,TBEN_C_DATA[121]);
   // Enable Diagnostics + In/Out Mapping: Swap All
   86: XIC(Common_Data.Port_in_Use.6)MOV(0,TBEN_C_DATA[121])MOV(3,TBEN_C_DATA[122])MOV(3,TBEN_C_DATA[123]);
   // Deactivate Diagnostics for unused port
   87: XIO(Common_Data.Port_in_Use.7)MOV(3,TBEN_C_DATA[137]);
   // Enable Diagnostics + In/Out Mapping: Swap All
   88: XIC(Common_Data.Port_in_Use.7)MOV(0,TBEN_C_DATA[137])MOV(3,TBEN_C_DATA[138])MOV(3,TBEN_C_DATA[139]);
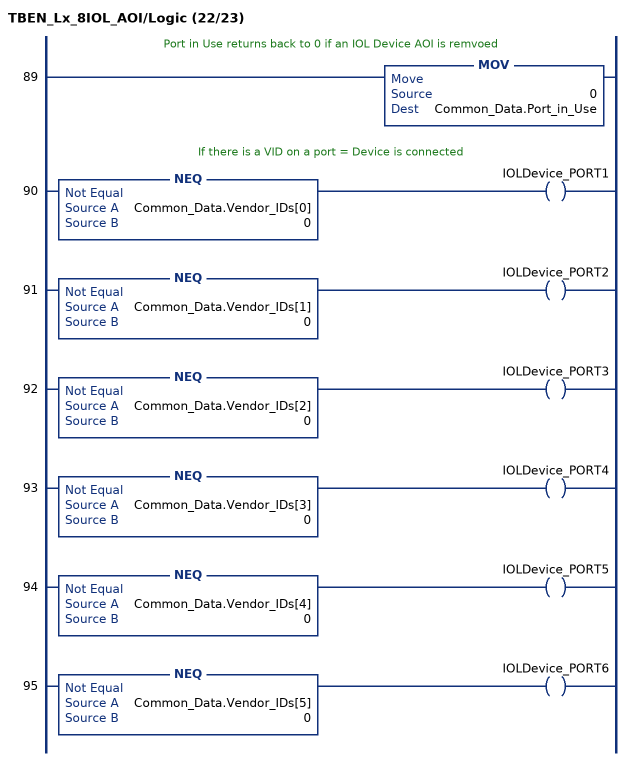
   // Port in Use returns back to 0 if an IOL Device AOI is remvoed
   89: MOV(0,Common_Data.Port_in_Use);
   // If there is a VID on a port = Device is connected
   90: NEQ(Common_Data.Vendor_IDs[0],0)OTE(IOLDevice_PORT1);
   91: NEQ(Common_Data.Vendor_IDs[1],0)OTE(IOLDevice_PORT2);
   92: NEQ(Common_Data.Vendor_IDs[2],0)OTE(IOLDevice_PORT3);
   93: NEQ(Common_Data.Vendor_IDs[3],0)OTE(IOLDevice_PORT4);
   94: NEQ(Common_Data.Vendor_IDs[4],0)OTE(IOLDevice_PORT5);
   95: NEQ(Common_Data.Vendor_IDs[5],0)OTE(IOLDevice_PORT6);
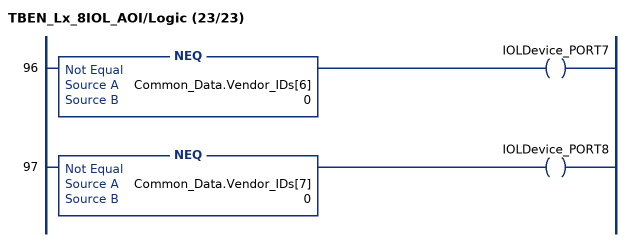
   96: NEQ(Common_Data.Vendor_IDs[6],0)OTE(IOLDevice_PORT7);
   97: NEQ(Common_Data.Vendor_IDs[7],0)OTE(IOLDevice_PORT8);
END_ROUTINE
